PROGRAM MAIN
VAR
	fbColor	: FB_Color;
END_VAR

END_PROGRAM

(* stored: Version 1.1.0.1, ProductVersion 3.1.4024.11
   POU MAIN: Id {f911f255-8ed5-4d04-bfb3-f2d3f2b160eb}, SpecialFunc None *)
